PROGRAM DomeLowLevelControl
VAR_INPUT
	enable : BOOL;
END_VAR
VAR
	Inverter_Enable:	BOOL;
	Inverter_Velocity:	UINT;
END_VAR

(* source: https://infosys.beckhoff.de/english.php?content=../content/1033/tcplclib_tc2_system/18014399220202635.html&id= *)

IF GVL_Dome.bVeloHigh THEN
	// High Speed
	Inverter_Velocity := 32767;
	Inverter_Enable := enable;
ELSIF GVL_Dome.bVeloLow THEN
	// low speed
	Inverter_Velocity := 10000;
	Inverter_Enable := enable;
ELSIF GVL_Dome.bBreak THEN
	// breaking (halt)
	Inverter_Velocity := 0;
	Inverter_Enable := FALSE;
ELSE
	// default
	Inverter_Velocity := 0;
	Inverter_Enable := FALSE;
END_IF

GVL_Dome.Inverter_DirectionMinus := GVL_Dome.bDirectionPlus;
GVL_Dome.Inverter_Enable := Inverter_Enable;
GVL_Dome.Inverter_Velocity := Inverter_Velocity;

END_PROGRAM

(* stored: Version 1.1.0.1, ProductVersion 3.1.4024.9
   POU DomeLowLevelControl: Id {5043f649-b650-4559-92ff-7f85fab560c6}, SpecialFunc None *)
